FUNCTION_BLOCK TTestSuite EXTENDS tcl_UnitTestBaseClasses.TTestSuite // Used to make TTestSuite accesible via this library

END_FUNCTION_BLOCK

(* stored: Version 1.1.0.1, ProductVersion 3.1.4024.4
   POU TTestSuite: Id {784949de-5ba9-4ac4-bfde-1c895feeccc0}, SpecialFunc None *)
